# EPICS autosave request: softglue/softGlueApp/Db/softGlue_settings.req
file softGlue_SignalShow_settings.req P=$(P) H=$(H)
file softGlue_FPGAContent_settings.req P=$(P) H=$(H)
file softGlue_FPGAInt_settings.req P=$(P) H=$(H)
file softGlue_convenience_settings.req P=$(P) H=$(H)
# If you've loaded softGlue_FPGAContent_octupole_settings.db, uncomment
# the following line.
#file softGlue_FPGAContent_octupole_settings.req P=$(P) H=$(H)
